(* PLC project Unnamed, Unknown Unnamed 1 *)
(* stored: creationDateTime 2021-02-24T10:39:13, modificationDateTime 2022-08-17T13:50:20 *)

PROGRAM program0
  VAR
    LED_PIN : BOOL;
    INIT_SUCCESS : BOOL;
    TON0 : TON;
    TOF0 : TOF;
    P1AM_INIT0 : P1AM_INIT;
    P1_16CDR0 : P1_16CDR;
  END_VAR

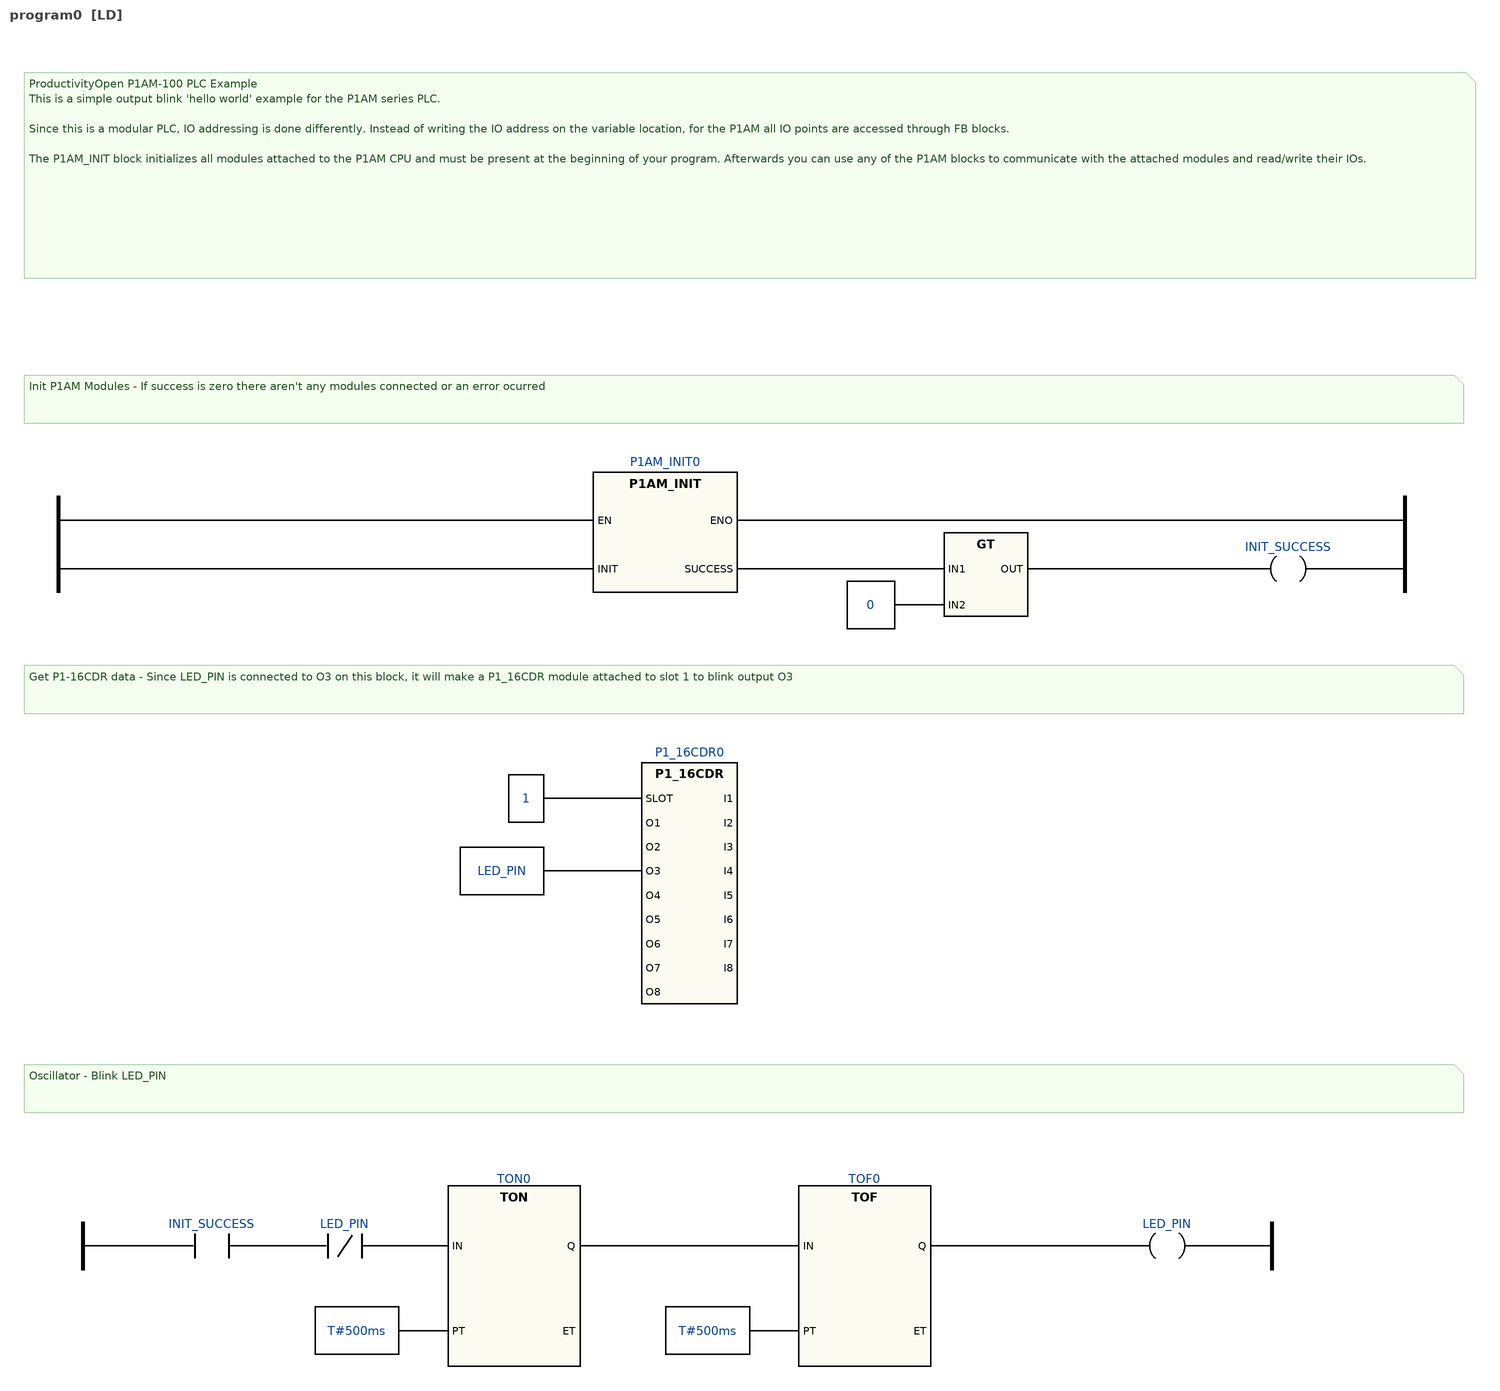
(* LD diagram, written out as Structured Text *)
(* ProductivityOpen P1AM-100 PLC Example
This is a simple output blink 'hello world' example for the P1AM series PLC. 

Since this is a modular PLC, IO addressing is done differently. Instead of writing the IO address on the variable location, for the P1AM all IO points are accessed through FB blocks. 

The P1AM_INIT block initializes all modules attached to the P1AM CPU and must be present at the beginning of your program. Afterwards you can use any of the P1AM blocks to communicate with the attached modules and read/write their IOs. *)
(* Init P1AM Modules - If success is zero there aren't any modules connected or an error ocurred *)
P1AM_INIT0(INIT := TRUE);
INIT_SUCCESS := P1AM_INIT0.SUCCESS > 0;
(* Get P1-16CDR data - Since LED_PIN is connected to O3 on this block, it will make a P1_16CDR module attached to slot 1 to blink output O3 *)
(* Oscillator - Blink LED_PIN *)
TON0(IN := INIT_SUCCESS AND NOT LED_PIN, PT := T#500ms);
TOF0(IN := TON0.Q, PT := T#500ms);
LED_PIN := TOF0.Q;
P1_16CDR0(SLOT := 1, O3 := LED_PIN);
END_PROGRAM

CONFIGURATION Config0
  RESOURCE Res0 ON PLC
    TASK task0(INTERVAL := T#20ms, PRIORITY := 0);
    PROGRAM instance0 WITH task0 : program0;
  END_RESOURCE
END_CONFIGURATION
